FUNCTION_BLOCK App3_SeparatorLevel (* Composite Function Block Type *)
  (* Standard: 61499-2 *)
  (* Version 0.0, 2018-11-06, 4DIAC-IDE, 4DIAC-Consortium *)
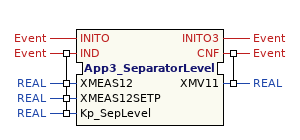
  EVENT_INPUT
    INITO; (* Initialization Request *)
    IND WITH XMEAS12, XMEAS12SETP, Kp_SepLevel; (* Normal Execution Request *)
  END_EVENT
  EVENT_OUTPUT
    INITO3; (* Initialization Confirm *)
    CNF WITH XMV11; (* Execution Confirmation *)
  END_EVENT
  VAR_INPUT
    XMEAS12 : REAL;
    XMEAS12SETP : REAL;
    Kp_SepLevel : REAL;
  END_VAR
  VAR_OUTPUT
    XMV11 : REAL;
  END_VAR
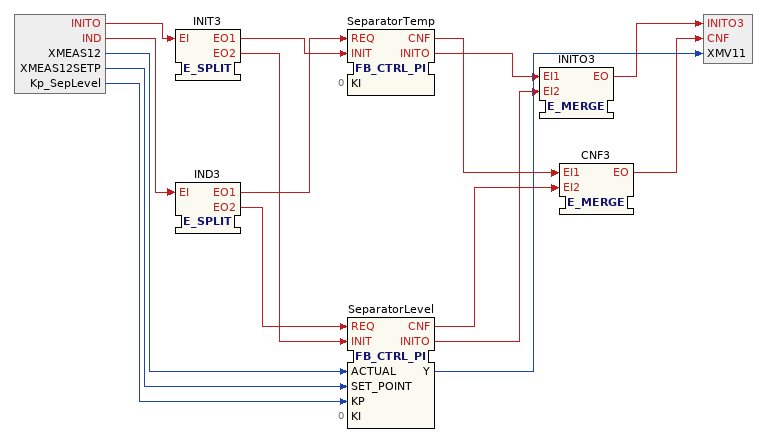
  FBS
    IND3 : E_SPLIT;
    CNF3 : E_MERGE;
    SeparatorTemp : FB_CTRL_PI(KI := 0);
    SeparatorLevel : FB_CTRL_PI(KI := 0);
    INIT3 : E_SPLIT;
    INITO3 : E_MERGE;
  END_FBS
  EVENT_CONNECTIONS
    IND3.EO1 TO SeparatorTemp.REQ;
    IND3.EO2 TO SeparatorLevel.REQ;
    SeparatorTemp.CNF TO CNF3.EI1;
    SeparatorLevel.CNF TO CNF3.EI2;
    CNF3.EO TO CNF;
    IND TO IND3.EI;
    INITO TO INIT3.EI;
    INIT3.EO1 TO SeparatorTemp.INIT;
    INIT3.EO2 TO SeparatorLevel.INIT;
    SeparatorTemp.INITO TO INITO3.EI1;
    SeparatorLevel.INITO TO INITO3.EI2;
    INITO3.EO TO INITO3;
  END_CONNECTIONS
  DATA_CONNECTIONS
    SeparatorLevel.Y TO XMV11;
    XMEAS12 TO SeparatorLevel.ACTUAL;
    XMEAS12SETP TO SeparatorLevel.SET_POINT;
    Kp_SepLevel TO SeparatorLevel.KP;
  END_CONNECTIONS
END_FUNCTION_BLOCK
